SYSTEM Xplus3Matlab
  (* Version 1.0, Author, 4DIAC-Consortium *)
  APPLICATION Xplus3MatlabApp
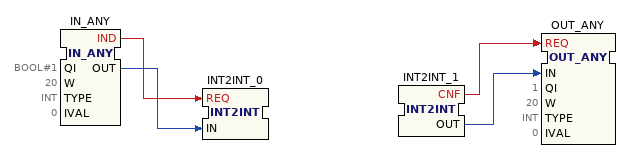
    FBS
      OUT_ANY : OUT_ANY(QI := 1, W := 20, TYPE := INT, IVAL := 0);
      INT2INT_0 : INT2INT;
      IN_ANY : IN_ANY(QI := BOOL#1, W := 20, TYPE := INT, IVAL := 0);
      INT2INT_1 : INT2INT;
    END_FBS
    EVENT_CONNECTIONS
      INT2INT_1.CNF TO OUT_ANY.REQ;
      IN_ANY.IND TO INT2INT_0.REQ;
    END_CONNECTIONS
    DATA_CONNECTIONS
      INT2INT_1.OUT TO OUT_ANY.IN;
      IN_ANY.OUT TO INT2INT_0.IN;
    END_CONNECTIONS
  END_APPLICATION
  DEVICE FBRT_WINDOW : FBRT_WINDOW(MGR_ID := "localhost:61499")
    {SET_ATTRIBUTE(Profile, HOLOBLOC)}
    RESOURCE PANEL_RESOURCE : PANEL_RESOURCE
    END_RESOURCE
  END_DEVICE
  DEVICE FORTE_PC : FORTE_PC(MGR_ID := "localhost:61499")
    {SET_ATTRIBUTE(Profile, HOLOBLOC)}
    RESOURCE EMB_RES : EMB_RES
    END_RESOURCE
  END_DEVICE
  SEGMENTS
    Ethernet : Ethernet;
  END_SEGMENTS
END_SYSTEM
